PROGRAM PRG_Automatic
VAR
	nState				: INT;
	rtExecute			: R_TRIG;
	rtAbort				: R_TRIG;
	nNumberOfParts		: INT;
	nCounter			: INT;
	i					: INT;
	bNotBusy			: BOOL;
	bError				: bool;
END_VAR
VAR CONSTANT
	Z_UP				: LREAL := 200.0;
	Z_DOWN				: LREAL := 0.0;
	X1					: LREAL := 500.0;
	Y1					: LREAL := 500.0;
	X2					: LREAL := -300.0;
	Y2					: LREAL := -300.0;
	NUMBER_OF_PARTS		: ARRAY[0..2] OF INT := [3, 5, 10];
END_VAR

rtExecute(CLK:=GVL.stProgramCtrl.bExecute);
rtAbort(CLK:=GVL.stProgramCtrl.bAbort);
GVL.stProgramCtrl.bExecute R= GVL.bReset;
GVL.stProgramCtrl.bAbort R= GVL.bReset;
IF nState>0 AND (rtAbort.Q OR GVL.bReset OR GVL.bError) THEN
	bError := GVL.bError;
	nState := -1;
END_IF

CASE nState OF
	-1:		// Abort
		bNotBusy := TRUE;	
		FOR i:=1 TO 3 DO
			GVL.aMoveAbsCtrl[i].bAbort := TRUE;
			bNotBusy := bNotBusy AND NOT GVL.aMoveAbsState[i].bBusy;
		END_FOR
		IF bNotBusy THEN
			FOR i:=1 TO 3 DO
				GVL.aMoveAbsCtrl[i].bExecute := FALSE;
				GVL.aMoveAbsCtrl[i].bAbort := FALSE;
			END_FOR
			GVL.stProgramState.bBusy := FALSE;
			GVL.stProgramState.bAborted := NOT bError;
			GVL.stProgramState.bError := bError;
			nState := 0;
		END_IF
		
	0:		// Idle
		IF rtExecute.Q THEN
			nNumberOfParts := NUMBER_OF_PARTS[GVL.nProgramNo];
			nCounter := 0;
			GVL.stProgramState.bBusy := TRUE;
			nState := nState + 1;
		ELSIF NOT GVL.stProgramCtrl.bExecute THEN
			bError := FALSE;
			GVL.stProgramState.nErrorId := 0;
			GVL.stProgramState.bError := FALSE;
			GVL.stProgramState.bBusy := FALSE;
			GVL.stProgramState.bAborted := FALSE;
			GVL.stProgramState.bDone := FALSE;
		END_IF
		
	1:		// Open Gripper
		GVL.stGripperCtrl.bReset := TRUE;
		IF GVL.stGripperState.bDone AND GVL.stGripperState.bOff THEN
			GVL.stGripperCtrl.bReset := FALSE;
			nState := nState + 1;
		ELSIF GVL.stGripperState.bError THEN
			bError := TRUE;
			GVL.stProgramState.nErrorId := INT_TO_UDINT(nState);
			nState := -1;
		END_IF
		
	2:		// Move Z up
		GVL.aTargetPos[3] := Z_UP;
		GVL.aMoveAbsCtrl[3].bExecute := TRUE;
		IF GVL.aMoveAbsState[3].bDone THEN
			GVL.aMoveAbsCtrl[3].bExecute := FALSE;
			nState := nState + 1;
		ELSIF GVL.aMoveAbsState[3].bError OR GVL.aMoveAbsState[3].bAborted THEN
			bError := TRUE;
			GVL.stProgramState.nErrorId := INT_TO_UDINT(nState);
			nState := -1;
		END_IF
		
	3:		// Move to Pos 1
		GVL.aTargetPos[1] := X1;
		GVL.aTargetPos[2] := Y1;
		GVL.aMoveAbsCtrl[1].bExecute := TRUE;
		GVL.aMoveAbsCtrl[2].bExecute := TRUE;
		IF GVL.aMoveAbsState[1].bDone AND GVL.aMoveAbsState[2].bDone THEN
			GVL.aMoveAbsCtrl[1].bExecute := FALSE;
			GVL.aMoveAbsCtrl[2].bExecute := FALSE;
			nState := nState + 1;
		ELSIF GVL.aMoveAbsState[1].bError OR GVL.aMoveAbsState[1].bAborted OR 
			  GVL.aMoveAbsState[2].bError OR GVL.aMoveAbsState[2].bAborted THEN
			bError := TRUE;
			GVL.stProgramState.nErrorId := INT_TO_UDINT(nState);
			nState := -1;
		END_IF
		
	4:		// Move Z down
		GVL.aTargetPos[3] := Z_DOWN;
		GVL.aMoveAbsCtrl[3].bExecute := TRUE;
		IF GVL.aMoveAbsState[3].bDone THEN
			GVL.aMoveAbsCtrl[3].bExecute := FALSE;
			nState := nState + 1;
		ELSIF GVL.aMoveAbsState[3].bError OR GVL.aMoveAbsState[3].bAborted THEN
			bError := TRUE;
			GVL.stProgramState.nErrorId := INT_TO_UDINT(nState);
			nState := -1;
		END_IF
		
	5:		// Close Gripper
		GVL.stGripperCtrl.bSet := TRUE;
		IF GVL.stGripperState.bDone AND GVL.stGripperState.bOn THEN
			GVL.stGripperCtrl.bSet := FALSE;
			nState := nState + 1;
		ELSIF GVL.stGripperState.bError THEN
			bError := TRUE;
			GVL.stProgramState.nErrorId := INT_TO_UDINT(nState);
			nState := -1;
		END_IF
		
	6:		// Move Z up
		GVL.aTargetPos[3] := Z_UP;
		GVL.aMoveAbsCtrl[3].bExecute := TRUE;
		IF GVL.aMoveAbsState[3].bDone THEN
			GVL.aMoveAbsCtrl[3].bExecute := FALSE;
			nState := nState + 1;
		ELSIF GVL.aMoveAbsState[3].bError OR GVL.aMoveAbsState[3].bAborted THEN
			bError := TRUE;
			GVL.stProgramState.nErrorId := INT_TO_UDINT(nState);
			nState := -1;
		END_IF
		
	7:		// Move to Pos 2
		GVL.aTargetPos[1] := X2;
		GVL.aTargetPos[2] := Y2;
		GVL.aMoveAbsCtrl[1].bExecute := TRUE;
		GVL.aMoveAbsCtrl[2].bExecute := TRUE;
		IF GVL.aMoveAbsState[1].bDone AND GVL.aMoveAbsState[2].bDone THEN
			GVL.aMoveAbsCtrl[1].bExecute := FALSE;
			GVL.aMoveAbsCtrl[2].bExecute := FALSE;
			nState := nState + 1;
		ELSIF GVL.aMoveAbsState[1].bError OR GVL.aMoveAbsState[1].bAborted OR 
			  GVL.aMoveAbsState[2].bError OR GVL.aMoveAbsState[2].bAborted THEN			
			bError := TRUE;
			GVL.stProgramState.nErrorId := INT_TO_UDINT(nState);
			nState := -1;
		END_IF
		
	8:		// Move Z down
		GVL.aTargetPos[3] := Z_DOWN;
		GVL.aMoveAbsCtrl[3].bExecute := TRUE;
		IF GVL.aMoveAbsState[3].bDone THEN
			GVL.aMoveAbsCtrl[3].bExecute := FALSE;
			nState := nState + 1;
		ELSIF GVL.aMoveAbsState[3].bError OR GVL.aMoveAbsState[3].bAborted THEN
			bError := TRUE;
			GVL.stProgramState.nErrorId := INT_TO_UDINT(nState);
			nState := -1;
		END_IF
		
	9:		// Open Gripper
		GVL.stGripperCtrl.bReset := TRUE;
		IF GVL.stGripperState.bDone AND GVL.stGripperState.bOff THEN
			GVL.stGripperCtrl.bReset := FALSE;
			nState := nState + 1;
			nCounter := nCounter + 1;
		ELSIF GVL.stGripperState.bError THEN
			bError := TRUE;
			GVL.stProgramState.nErrorId := INT_TO_UDINT(nState);
			nState := -1;
		END_IF
		
	10:
		IF nCounter = nNumberOfParts THEN
			GVL.stProgramState.bBusy := FALSE;
			GVL.stProgramState.bDone := TRUE;
			nState := 0;
		ELSE
			nState := 1;
		END_IF
		
	
END_CASE

GVL.nProgramStep := nState + 1;

IF GVL.stProgramState.bError THEN
	GVL.nProgramState := 4;
ELSIF GVL.stProgramState.bAborted THEN
	GVL.nProgramState := 3;
ELSIF GVL.stProgramState.bDone THEN
	GVL.nProgramState := 2;
ELSIF GVL.stProgramState.bBusy THEN
	GVL.nProgramState := 1;
ELSE
	GVL.nProgramState := 0;
END_IF

END_PROGRAM

(* stored: Version 1.1.0.1, ProductVersion 3.1.4024.15
   POU PRG_Automatic: Id {738e971c-cbb0-4d55-88ba-bb46eb819197}, SpecialFunc None *)
